INTERFACE I_LightBase EXTENDS __SYSTEM.IQueryInterface

PROPERTY ID : USINT
GET
END_GET
SET
END_SET
END_PROPERTY

PROPERTY PUBLIC State : BOOL
GET
END_GET
SET
END_SET
END_PROPERTY

METHOD Toggle
END_METHOD

METHOD TurnOFF
END_METHOD

METHOD TurnON
END_METHOD

END_INTERFACE

(* stored: Version 1.1.0.1, ProductVersion 3.1.4024.12
   Itf I_LightBase: Id {39719b6d-833f-4ef2-afd1-42b91cf29e24}
   Property ID: Id {0d156c20-f81d-4493-a12c-e0789cfeb86e}
   Get Get: Id {a17ff519-695b-434f-b223-8163925c467f}
   Set Set: Id {c4a90f44-115b-4e0b-92be-d515173e4870}
   Property State: Id {0576a3eb-e9ad-4a58-9e4d-623558461fc4}
   Get Get: Id {d8fedb75-476f-42eb-b9a8-36b0617fcd1e}
   Set Set: Id {a032fb47-539c-4f1a-abf4-2b58e4b44394}
   Method Toggle: Id {2041c29b-f883-4122-894e-14e4e342b6dd}
   Method TurnOFF: Id {996e40d5-a823-4391-8fc0-3f8b18fe357e}
   Method TurnON: Id {a4e99652-e0d2-4c30-a533-09b77f612dd9} *)
